// TwinCAT 3 PLC project RTNNI
// Title: Real-Time Neural Network Inference
// Company: ISW
// Author: Zexu Zhou, Christoph Hinze, Haijia Xu, Armin Lechler, Alexander Verl
// ProjectVersion: 0.1
// ProgramVersion: 3.1.4024.0
// libraries:
//   Tc2_Standard, * (Beckhoff Automation GmbH)
//   Tc2_System, * (Beckhoff Automation GmbH)
//   Tc2_Utilities, * (Beckhoff Automation GmbH)
//   Tc3_Module, * (Beckhoff Automation GmbH)
// project tree:
//   DUTs/ act_type.TcDUT, Layer.TcDUT
//   / PlcTask.TcTTO (not stored)
//   POUs/activation function/ F_exponential.TcPOU (not stored), F_relu.TcPOU (not stored), F_selu.TcPOU (not stored), F_sigmoid.TcPOU (not stored), F_silu.TcPOU, F_softplus.TcPOU (not stored), F_softsign.TcPOU (not stored), F_tanh.TcPOU (not stored)
//   POUs/ FB_LoadWeights.TcPOU (not stored), F_ForwardPropagation.TcPOU (not stored)
//   POUs/math/ F_Dot.TcPOU (not stored)
//   POUs/normalization/ F_denormalization.TcPOU (not stored), F_normalization.TcPOU (not stored), F_NormalizationLayer.TcPOU (not stored)

// ---- DUTs/act_type.TcDUT
{attribute 'qualified_only'}
{attribute 'strict'}
TYPE act_type :
(
	linear := 0,
	relu :=1,
	tanh :=2,
	sigmoid :=3,
	softplus := 4,
	softsign := 5,
	silu := 6,
	selu := 7,
	exponential := 8
);
END_TYPE

// ---- DUTs/Layer.TcDUT
TYPE Layer :
STRUCT
	num_neurons : UINT;
	activation : act_type;
	pointer_weight: POINTER TO LREAL;
	pointer_bias: POINTER TO LREAL;
END_STRUCT
END_TYPE

// ---- POUs/activation function/F_silu.TcPOU
FUNCTION F_silu : lreal
VAR_INPUT
	x : LREAL;
END_VAR

IF x > 1E2 THEN
	F_silu := x;
ELSIF x < -1E2 THEN
	F_silu := 0;
ELSE
	F_silu := x / (1 + EXP(-x));
END_IF

END_FUNCTION
